TYPE TcaSafetyGateConfig :
STRUCT
	
END_STRUCT
END_TYPE

(* stored: Version 1.1.0.1
   DUT TcaSafetyGateConfig: Id {15c070ef-8cc3-4dbc-b523-8854f802b997} *)
